// TIA Portal V16 export
// export: Created 2024-05-10T06:46:41.2212007Z, ExportSetting WithDefaults, DisplayName Totally Integrated Automation Portal, DisplayVersion V16, DisplayName TIA Portal Version Control Interface, DisplayVersion V16, DisplayName TIA Portal Openness, DisplayVersion V16, DisplayName STEP 7 Professional, DisplayVersion V16, DisplayName STEP 7 Safety, DisplayVersion V16, DisplayName WinCC Professional, DisplayVersion V16
FUNCTION_BLOCK "K07_轴组"   // FB7, LAD
{ S7_Optimized_Access := 'TRUE' }
VERSION : 0.1
// stored: AutoNumber false, IsIECCheckEnabled false, IsRetainMemResEnabled false, MemoryReserve 100, SetENOAutomatically false, UDAEnableTagReadback false
   VAR
      Axis1Write { S7_SetPoint := 'True'} : "F121_SinaParaWrite(SV660F)";   // 轴1参数
      Axis1Pos { S7_SetPoint := 'True'} : "F120_SinaPos(SV660F)";   // 轴1定位
   END_VAR
   VAR_TEMP   // added for the SCL form of the ladder/FBD networks
      _w1 : Bool;
      _w2 : Bool;
      _w3 : Bool;
      _w4 : Bool;
      _w5 : Bool;
      _w6 : Bool;
      _w7 : Bool;
      _w8 : Bool;
      _w9 : Bool;
   END_VAR
BEGIN

REGION Network 1: 轴1参数
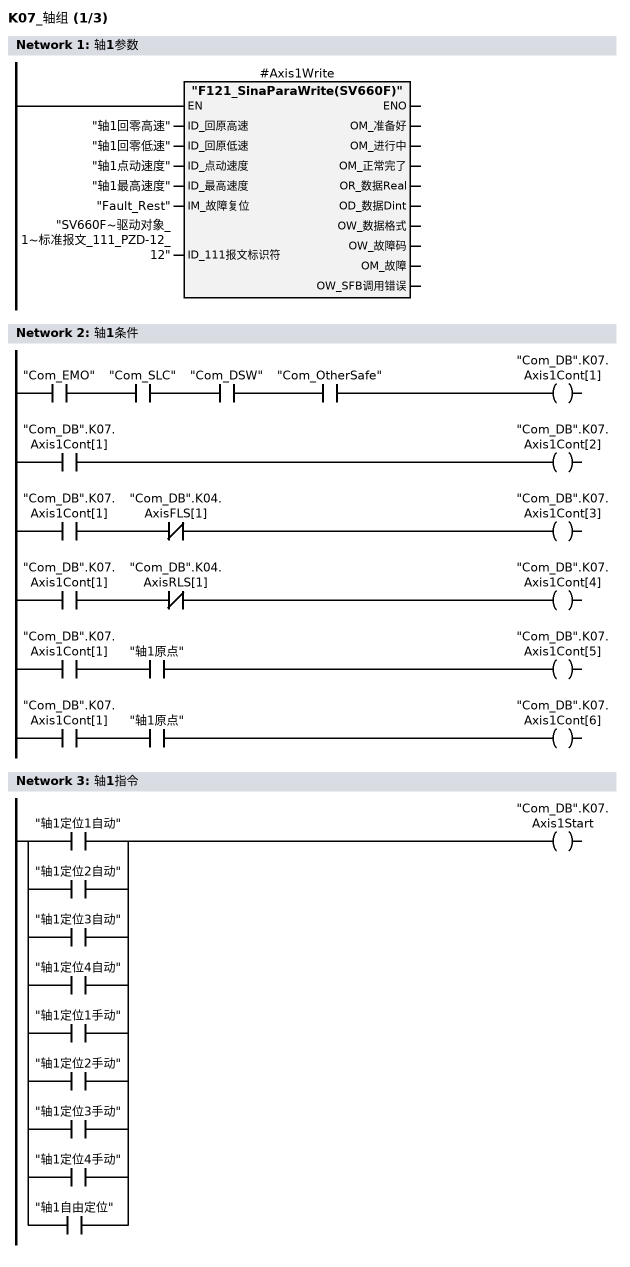
   RUNG wire#powerrail
      #Axis1Write(ID_回原高速 := "轴1回零高速", ID_回原低速 := "轴1回零低速", ID_点动速度 := "轴1点动速度", ID_最高速度 := "轴1最高速度", IM_故障复位 := "Fault_Rest", ID_111报文标识符 := "SV660F~驱动对象_1~标准报文_111_PZD-12_12", OM_准备好 =>, OM_进行中 =>, OM_正常完了 =>, OR_数据Real =>, OD_数据Dint =>, OW_数据格式 =>, OW_故障码 =>, OM_故障 =>, OW_SFB调用错误 =>)
   END_RUNG
   // the same network as SCL:
   #Axis1Write(ID_回原高速 := "轴1回零高速",   // "F121_SinaParaWrite(SV660F)"
               ID_回原低速 := "轴1回零低速",
               ID_点动速度 := "轴1点动速度",
               ID_最高速度 := "轴1最高速度",
               IM_故障复位 := "Fault_Rest",
               ID_111报文标识符 := "SV660F~驱动对象_1~标准报文_111_PZD-12_12");
END_REGION

REGION Network 2: 轴1条件
   RUNG wire#powerrail
      Contact( "Com_EMO" )
      Contact( "Com_SLC" )
      Contact( "Com_DSW" )
      Contact( "Com_OtherSafe" )
      Coil( "Com_DB".K07.Axis1Cont[1] )
   END_RUNG
   RUNG wire#powerrail
      Contact( "Com_DB".K07.Axis1Cont[1] )
      Coil( "Com_DB".K07.Axis1Cont[2] )
   END_RUNG
   RUNG wire#powerrail
      Contact( "Com_DB".K07.Axis1Cont[1] )
      I_Contact( "Com_DB".K04.AxisFLS[1] )
      Coil( "Com_DB".K07.Axis1Cont[3] )
   END_RUNG
   RUNG wire#powerrail
      Contact( "Com_DB".K07.Axis1Cont[1] )
      I_Contact( "Com_DB".K04.AxisRLS[1] )
      Coil( "Com_DB".K07.Axis1Cont[4] )
   END_RUNG
   RUNG wire#powerrail
      Contact( "Com_DB".K07.Axis1Cont[1] )
      Contact( "轴1原点" )
      Coil( "Com_DB".K07.Axis1Cont[5] )
   END_RUNG
   RUNG wire#powerrail
      Contact( "Com_DB".K07.Axis1Cont[1] )
      Contact( "轴1原点" )
      Coil( "Com_DB".K07.Axis1Cont[6] )
   END_RUNG
   // the same network as SCL:
   "Com_DB".K07.Axis1Cont[1] := "Com_EMO" AND "Com_SLC" AND "Com_DSW" AND "Com_OtherSafe";
   "Com_DB".K07.Axis1Cont[2] := "Com_DB".K07.Axis1Cont[1];
   "Com_DB".K07.Axis1Cont[3] := "Com_DB".K07.Axis1Cont[1] AND NOT "Com_DB".K04.AxisFLS[1];
   "Com_DB".K07.Axis1Cont[4] := "Com_DB".K07.Axis1Cont[1] AND NOT "Com_DB".K04.AxisRLS[1];
   "Com_DB".K07.Axis1Cont[5] := "Com_DB".K07.Axis1Cont[1] AND "轴1原点";
   "Com_DB".K07.Axis1Cont[6] := "Com_DB".K07.Axis1Cont[1] AND "轴1原点";
END_REGION

REGION Network 3: 轴1指令
   RUNG wire#powerrail
      Contact( "轴1定位1自动" )
      wire#w1
      Coil( "Com_DB".K07.Axis1Start )
   END_RUNG
   RUNG wire#powerrail
      Contact( "轴1定位2自动" )
   END_RUNG wire#w1
   RUNG wire#powerrail
      Contact( "轴1定位3自动" )
   END_RUNG wire#w1
   RUNG wire#powerrail
      Contact( "轴1定位4自动" )
   END_RUNG wire#w1
   RUNG wire#powerrail
      Contact( "轴1定位1手动" )
   END_RUNG wire#w1
   RUNG wire#powerrail
      Contact( "轴1定位2手动" )
   END_RUNG wire#w1
   RUNG wire#powerrail
      Contact( "轴1定位3手动" )
   END_RUNG wire#w1
   RUNG wire#powerrail
      Contact( "轴1定位4手动" )
   END_RUNG wire#w1
   RUNG wire#powerrail
      Contact( "轴1自由定位" )
   END_RUNG wire#w1
   // the same network as SCL:
   "Com_DB".K07.Axis1Start := "轴1定位1自动" OR "轴1定位2自动" OR "轴1定位3自动" OR "轴1定位4自动" OR "轴1定位1手动" OR "轴1定位2手动" OR "轴1定位3手动" OR "轴1定位4手动" OR "轴1自由定位";
END_REGION

REGION Network 4: 轴1位置速度
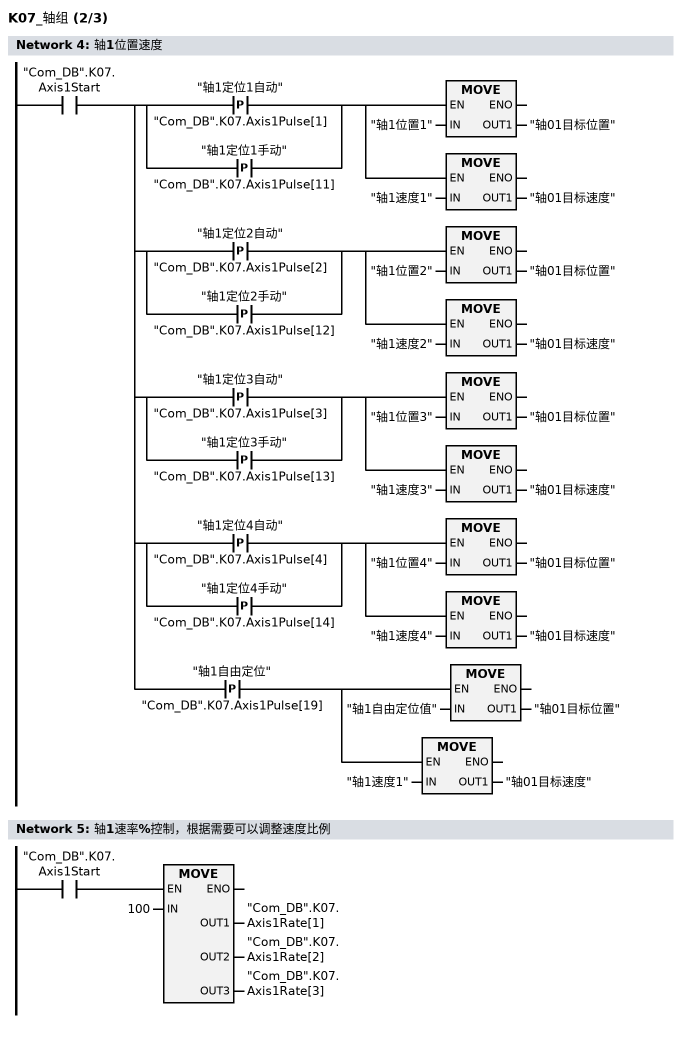
   RUNG wire#powerrail
      Contact( "Com_DB".K07.Axis1Start )
      wire#w1
      P_Contact(operand := "轴1定位1自动", bit := "Com_DB".K07.Axis1Pulse[1])
      wire#w2
      Move(in := "轴1位置1", out1 => "轴01目标位置")
   END_RUNG
   RUNG wire#w1
      P_Contact(operand := "轴1定位1手动", bit := "Com_DB".K07.Axis1Pulse[11])
   END_RUNG wire#w2
   RUNG wire#w2
      Move(in := "轴1速度1", out1 => "轴01目标速度")
   END_RUNG
   RUNG wire#w1
      P_Contact(operand := "轴1定位2自动", bit := "Com_DB".K07.Axis1Pulse[2])
      wire#w3
      Move(in := "轴1位置2", out1 => "轴01目标位置")
   END_RUNG
   RUNG wire#w1
      P_Contact(operand := "轴1定位2手动", bit := "Com_DB".K07.Axis1Pulse[12])
   END_RUNG wire#w3
   RUNG wire#w3
      Move(in := "轴1速度2", out1 => "轴01目标速度")
   END_RUNG
   RUNG wire#w1
      P_Contact(operand := "轴1定位3自动", bit := "Com_DB".K07.Axis1Pulse[3])
      wire#w4
      Move(in := "轴1位置3", out1 => "轴01目标位置")
   END_RUNG
   RUNG wire#w1
      P_Contact(operand := "轴1定位3手动", bit := "Com_DB".K07.Axis1Pulse[13])
   END_RUNG wire#w4
   RUNG wire#w4
      Move(in := "轴1速度3", out1 => "轴01目标速度")
   END_RUNG
   RUNG wire#w1
      P_Contact(operand := "轴1定位4自动", bit := "Com_DB".K07.Axis1Pulse[4])
      wire#w5
      Move(in := "轴1位置4", out1 => "轴01目标位置")
   END_RUNG
   RUNG wire#w1
      P_Contact(operand := "轴1定位4手动", bit := "Com_DB".K07.Axis1Pulse[14])
   END_RUNG wire#w5
   RUNG wire#w5
      Move(in := "轴1速度4", out1 => "轴01目标速度")
   END_RUNG
   RUNG wire#w1
      P_Contact(operand := "轴1自由定位", bit := "Com_DB".K07.Axis1Pulse[19])
      wire#w6
      Move(in := "轴1自由定位值", out1 => "轴01目标位置")
   END_RUNG
   RUNG wire#w6
      Move(in := "轴1速度1", out1 => "轴01目标速度")
   END_RUNG
   // the same network as SCL:
   #_w1 := "Com_DB".K07.Axis1Start AND "轴1定位1自动" AND NOT "Com_DB".K07.Axis1Pulse[1];   // rising edge of "轴1定位1自动"
   "Com_DB".K07.Axis1Pulse[1] := "轴1定位1自动";
   #_w2 := "Com_DB".K07.Axis1Start AND "轴1定位1手动" AND NOT "Com_DB".K07.Axis1Pulse[11];   // rising edge of "轴1定位1手动"
   "Com_DB".K07.Axis1Pulse[11] := "轴1定位1手动";
   IF #_w1 OR #_w2 THEN
       "轴01目标位置" := "轴1位置1";
       "轴01目标速度" := "轴1速度1";
   END_IF;
   #_w3 := "Com_DB".K07.Axis1Start AND "轴1定位2自动" AND NOT "Com_DB".K07.Axis1Pulse[2];   // rising edge of "轴1定位2自动"
   "Com_DB".K07.Axis1Pulse[2] := "轴1定位2自动";
   #_w4 := "Com_DB".K07.Axis1Start AND "轴1定位2手动" AND NOT "Com_DB".K07.Axis1Pulse[12];   // rising edge of "轴1定位2手动"
   "Com_DB".K07.Axis1Pulse[12] := "轴1定位2手动";
   IF #_w3 OR #_w4 THEN
       "轴01目标位置" := "轴1位置2";
       "轴01目标速度" := "轴1速度2";
   END_IF;
   #_w5 := "Com_DB".K07.Axis1Start AND "轴1定位3自动" AND NOT "Com_DB".K07.Axis1Pulse[3];   // rising edge of "轴1定位3自动"
   "Com_DB".K07.Axis1Pulse[3] := "轴1定位3自动";
   #_w6 := "Com_DB".K07.Axis1Start AND "轴1定位3手动" AND NOT "Com_DB".K07.Axis1Pulse[13];   // rising edge of "轴1定位3手动"
   "Com_DB".K07.Axis1Pulse[13] := "轴1定位3手动";
   IF #_w5 OR #_w6 THEN
       "轴01目标位置" := "轴1位置3";
       "轴01目标速度" := "轴1速度3";
   END_IF;
   #_w7 := "Com_DB".K07.Axis1Start AND "轴1定位4自动" AND NOT "Com_DB".K07.Axis1Pulse[4];   // rising edge of "轴1定位4自动"
   "Com_DB".K07.Axis1Pulse[4] := "轴1定位4自动";
   #_w8 := "Com_DB".K07.Axis1Start AND "轴1定位4手动" AND NOT "Com_DB".K07.Axis1Pulse[14];   // rising edge of "轴1定位4手动"
   "Com_DB".K07.Axis1Pulse[14] := "轴1定位4手动";
   IF #_w7 OR #_w8 THEN
       "轴01目标位置" := "轴1位置4";
       "轴01目标速度" := "轴1速度4";
   END_IF;
   #_w9 := "Com_DB".K07.Axis1Start AND "轴1自由定位" AND NOT "Com_DB".K07.Axis1Pulse[19];   // rising edge of "轴1自由定位"
   "Com_DB".K07.Axis1Pulse[19] := "轴1自由定位";
   IF #_w9 THEN
       "轴01目标位置" := "轴1自由定位值";
       "轴01目标速度" := "轴1速度1";
   END_IF;
END_REGION

REGION Network 5: 轴1速率%控制，根据需要可以调整速度比例
   RUNG wire#powerrail
      Contact( "Com_DB".K07.Axis1Start )
      Move(in := 100, out1 => "Com_DB".K07.Axis1Rate[1], out2 => "Com_DB".K07.Axis1Rate[2], out3 => "Com_DB".K07.Axis1Rate[3])
   END_RUNG
   // the same network as SCL:
   IF "Com_DB".K07.Axis1Start THEN
       "Com_DB".K07.Axis1Rate[1] := 100;
       "Com_DB".K07.Axis1Rate[2] := 100;
       "Com_DB".K07.Axis1Rate[3] := 100;
   END_IF;
END_REGION

REGION Network 6: 轴1Pos
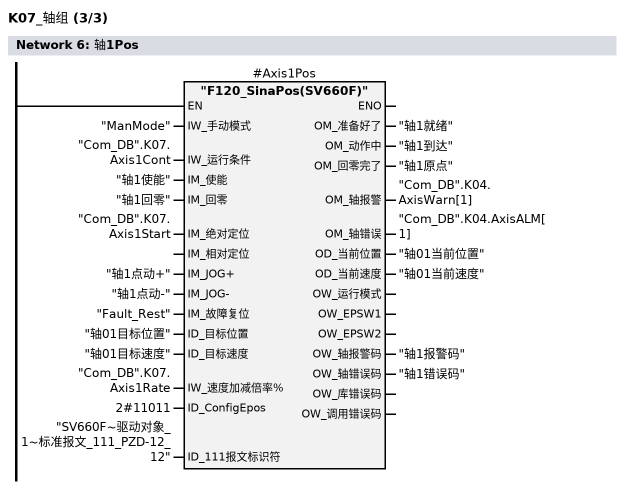
   RUNG wire#powerrail
      #Axis1Pos(IW_手动模式 := "ManMode", IW_运行条件 := "Com_DB".K07.Axis1Cont, IM_使能 := "轴1使能", IM_回零 := "轴1回零", IM_绝对定位 := "Com_DB".K07.Axis1Start, IM_相对定位 :=, "IM_JOG+" := "轴1点动+", "IM_JOG-" := "轴1点动-", IM_故障复位 := "Fault_Rest", ID_目标位置 := "轴01目标位置", ID_目标速度 := "轴01目标速度", "IW_速度加减倍率%" := "Com_DB".K07.Axis1Rate, ID_ConfigEpos := 2#11011, ID_111报文标识符 := "SV660F~驱动对象_1~标准报文_111_PZD-12_12", OM_准备好了 => "轴1就绪", OM_动作中 => "轴1到达", OM_回零完了 => "轴1原点", OM_轴报警 => "Com_DB".K04.AxisWarn[1], OM_轴错误 => "Com_DB".K04.AxisALM[1], OD_当前位置 => "轴01当前位置", OD_当前速度 => "轴01当前速度", OW_运行模式 =>, OW_EPSW1 =>, OW_EPSW2 =>, OW_轴报警码 => "轴1报警码", OW_轴错误码 => "轴1错误码", OW_库错误码 =>, OW_调用错误码 =>)
   END_RUNG
   // the same network as SCL:
   #Axis1Pos(IW_手动模式 := "ManMode",   // "F120_SinaPos(SV660F)"
             IW_运行条件 := "Com_DB".K07.Axis1Cont,
             IM_使能 := "轴1使能",
             IM_回零 := "轴1回零",
             IM_绝对定位 := "Com_DB".K07.Axis1Start,
             "IM_JOG+" := "轴1点动+",
             "IM_JOG-" := "轴1点动-",
             IM_故障复位 := "Fault_Rest",
             ID_目标位置 := "轴01目标位置",
             ID_目标速度 := "轴01目标速度",
             "IW_速度加减倍率%" := "Com_DB".K07.Axis1Rate,
             ID_ConfigEpos := 2#11011,
             ID_111报文标识符 := "SV660F~驱动对象_1~标准报文_111_PZD-12_12",
             OM_准备好了 => "轴1就绪",
             OM_动作中 => "轴1到达",
             OM_回零完了 => "轴1原点",
             OM_轴报警 => "Com_DB".K04.AxisWarn[1],
             OM_轴错误 => "Com_DB".K04.AxisALM[1],
             OD_当前位置 => "轴01当前位置",
             OD_当前速度 => "轴01当前速度",
             OW_轴报警码 => "轴1报警码",
             OW_轴错误码 => "轴1错误码");
END_REGION

REGION Network 7 (SCL): 轴1位置
   IF  ("轴1位置1"-2)<="轴01当前位置"
       AND ("轴1位置1"+2)>= "轴01当前位置"

   THEN
       "轴1定位1到位"           := TRUE         ;
   ELSE
       "轴1定位1到位" := FALSE;
   END_IF;// 

   IF ("轴1位置2" - 2) <= "轴01当前位置"
       AND ("轴1位置2" + 2) >= "轴01当前位置"

   THEN
       "轴1定位2到位" := TRUE;
   ELSE
       "轴1定位2到位" := FALSE;
   END_IF;

   IF ("轴1位置3" - 2) <= "轴01当前位置"
       AND ("轴1位置3" + 2) >= "轴01当前位置"

   THEN
       "轴1定位3到位" := TRUE;
   ELSE
       "轴1定位3到位" := FALSE;
   END_IF;

   IF ("轴1位置4" - 2) <= "轴01当前位置"
       AND ("轴1位置4" + 2) >= "轴01当前位置"

   THEN
       "轴1定位4到位" := TRUE;
   ELSE
       "轴1定位4到位" := FALSE;
   END_IF;
END_REGION

REGION Network 8: 轴1END
END_REGION
END_FUNCTION_BLOCK
